// TIA Portal V20 export
DATA_BLOCK "IdentMvHmi"   // DB214
// stored: MemoryReserve 100
   VAR
      unitIdentMv : Array[0.."NO_OF_UNITS"] of "typeEMIdentMv";
   END_VAR
BEGIN
   unitIdentMv[0].identMvEM[0..7].selectedUnit := 0;
   unitIdentMv[0].identMvEM[0..7].selectedEM := 0;
   unitIdentMv[0].identMvEM[0..7].mvReaderId := 0;
   unitIdentMv[0].identMvEM[0..7].numberOfMv := 0;
   unitIdentMv[0].identMvEM[0].mvReader[0..1].deviceName := WSTRING#'';
   unitIdentMv[0].identMvEM[1].mvReader[0..1].deviceName := WSTRING#'';
   unitIdentMv[0].identMvEM[2].mvReader[0..1].deviceName := WSTRING#'';
   unitIdentMv[0].identMvEM[3].mvReader[0..1].deviceName := WSTRING#'';
   unitIdentMv[0].identMvEM[4].mvReader[0..1].deviceName := WSTRING#'';
   unitIdentMv[0].identMvEM[5].mvReader[0..1].deviceName := WSTRING#'';
   unitIdentMv[0].identMvEM[6].mvReader[0..1].deviceName := WSTRING#'';
   unitIdentMv[0].identMvEM[7].mvReader[0..1].deviceName := WSTRING#'';
   unitIdentMv[0].identMvEM[0].mvReader[0..1].deviceType := WSTRING#'';
   unitIdentMv[0].identMvEM[1].mvReader[0..1].deviceType := WSTRING#'';
   unitIdentMv[0].identMvEM[2].mvReader[0..1].deviceType := WSTRING#'';
   unitIdentMv[0].identMvEM[3].mvReader[0..1].deviceType := WSTRING#'';
   unitIdentMv[0].identMvEM[4].mvReader[0..1].deviceType := WSTRING#'';
   unitIdentMv[0].identMvEM[5].mvReader[0..1].deviceType := WSTRING#'';
   unitIdentMv[0].identMvEM[6].mvReader[0..1].deviceType := WSTRING#'';
   unitIdentMv[0].identMvEM[7].mvReader[0..1].deviceType := WSTRING#'';
   unitIdentMv[0].identMvEM[0].mvReader[0..1].deviceId := 0;
   unitIdentMv[0].identMvEM[1].mvReader[0..1].deviceId := 0;
   unitIdentMv[0].identMvEM[2].mvReader[0..1].deviceId := 0;
   unitIdentMv[0].identMvEM[3].mvReader[0..1].deviceId := 0;
   unitIdentMv[0].identMvEM[4].mvReader[0..1].deviceId := 0;
   unitIdentMv[0].identMvEM[5].mvReader[0..1].deviceId := 0;
   unitIdentMv[0].identMvEM[6].mvReader[0..1].deviceId := 0;
   unitIdentMv[0].identMvEM[7].mvReader[0..1].deviceId := 0;
   unitIdentMv[0].identMvEM[0].mvReader[0..1].tagType := WSTRING#'';
   unitIdentMv[0].identMvEM[1].mvReader[0..1].tagType := WSTRING#'';
   unitIdentMv[0].identMvEM[2].mvReader[0..1].tagType := WSTRING#'';
   unitIdentMv[0].identMvEM[3].mvReader[0..1].tagType := WSTRING#'';
   unitIdentMv[0].identMvEM[4].mvReader[0..1].tagType := WSTRING#'';
   unitIdentMv[0].identMvEM[5].mvReader[0..1].tagType := WSTRING#'';
   unitIdentMv[0].identMvEM[6].mvReader[0..1].tagType := WSTRING#'';
   unitIdentMv[0].identMvEM[7].mvReader[0..1].tagType := WSTRING#'';
   unitIdentMv[0].identMvEM[0].mvReader[0..1].cameraMode := WSTRING#'';
   unitIdentMv[0].identMvEM[1].mvReader[0..1].cameraMode := WSTRING#'';
   unitIdentMv[0].identMvEM[2].mvReader[0..1].cameraMode := WSTRING#'';
   unitIdentMv[0].identMvEM[3].mvReader[0..1].cameraMode := WSTRING#'';
   unitIdentMv[0].identMvEM[4].mvReader[0..1].cameraMode := WSTRING#'';
   unitIdentMv[0].identMvEM[5].mvReader[0..1].cameraMode := WSTRING#'';
   unitIdentMv[0].identMvEM[6].mvReader[0..1].cameraMode := WSTRING#'';
   unitIdentMv[0].identMvEM[7].mvReader[0..1].cameraMode := WSTRING#'';
   unitIdentMv[0].identMvEM[0].mvReader[0..1].resultState := WSTRING#'';
   unitIdentMv[0].identMvEM[1].mvReader[0..1].resultState := WSTRING#'';
   unitIdentMv[0].identMvEM[2].mvReader[0..1].resultState := WSTRING#'';
   unitIdentMv[0].identMvEM[3].mvReader[0..1].resultState := WSTRING#'';
   unitIdentMv[0].identMvEM[4].mvReader[0..1].resultState := WSTRING#'';
   unitIdentMv[0].identMvEM[5].mvReader[0..1].resultState := WSTRING#'';
   unitIdentMv[0].identMvEM[6].mvReader[0..1].resultState := WSTRING#'';
   unitIdentMv[0].identMvEM[7].mvReader[0..1].resultState := WSTRING#'';
   unitIdentMv[0].identMvEM[0].mvReader[0..1].progNo := 0;
   unitIdentMv[0].identMvEM[1].mvReader[0..1].progNo := 0;
   unitIdentMv[0].identMvEM[2].mvReader[0..1].progNo := 0;
   unitIdentMv[0].identMvEM[3].mvReader[0..1].progNo := 0;
   unitIdentMv[0].identMvEM[4].mvReader[0..1].progNo := 0;
   unitIdentMv[0].identMvEM[5].mvReader[0..1].progNo := 0;
   unitIdentMv[0].identMvEM[6].mvReader[0..1].progNo := 0;
   unitIdentMv[0].identMvEM[7].mvReader[0..1].progNo := 0;
   unitIdentMv[0].identMvEM[0].mvReader[0..1].progNumberWrite := 0;
   unitIdentMv[0].identMvEM[1].mvReader[0..1].progNumberWrite := 0;
   unitIdentMv[0].identMvEM[2].mvReader[0..1].progNumberWrite := 0;
   unitIdentMv[0].identMvEM[3].mvReader[0..1].progNumberWrite := 0;
   unitIdentMv[0].identMvEM[4].mvReader[0..1].progNumberWrite := 0;
   unitIdentMv[0].identMvEM[5].mvReader[0..1].progNumberWrite := 0;
   unitIdentMv[0].identMvEM[6].mvReader[0..1].progNumberWrite := 0;
   unitIdentMv[0].identMvEM[7].mvReader[0..1].progNumberWrite := 0;
   unitIdentMv[0].identMvEM[0].mvReader[0..1].pushbutton := 16#0000;
   unitIdentMv[0].identMvEM[1].mvReader[0..1].pushbutton := 16#0000;
   unitIdentMv[0].identMvEM[2].mvReader[0..1].pushbutton := 16#0000;
   unitIdentMv[0].identMvEM[3].mvReader[0..1].pushbutton := 16#0000;
   unitIdentMv[0].identMvEM[4].mvReader[0..1].pushbutton := 16#0000;
   unitIdentMv[0].identMvEM[5].mvReader[0..1].pushbutton := 16#0000;
   unitIdentMv[0].identMvEM[6].mvReader[0..1].pushbutton := 16#0000;
   unitIdentMv[0].identMvEM[7].mvReader[0..1].pushbutton := 16#0000;
   unitIdentMv[0].identMvEM[0].mvReader[0..1].enablePushbutton := 16#0000;
   unitIdentMv[0].identMvEM[1].mvReader[0..1].enablePushbutton := 16#0000;
   unitIdentMv[0].identMvEM[2].mvReader[0..1].enablePushbutton := 16#0000;
   unitIdentMv[0].identMvEM[3].mvReader[0..1].enablePushbutton := 16#0000;
   unitIdentMv[0].identMvEM[4].mvReader[0..1].enablePushbutton := 16#0000;
   unitIdentMv[0].identMvEM[5].mvReader[0..1].enablePushbutton := 16#0000;
   unitIdentMv[0].identMvEM[6].mvReader[0..1].enablePushbutton := 16#0000;
   unitIdentMv[0].identMvEM[7].mvReader[0..1].enablePushbutton := 16#0000;
   unitIdentMv[0].identMvEM[0].mvReader[0..1].status := 16#0000;
   unitIdentMv[0].identMvEM[1].mvReader[0..1].status := 16#0000;
   unitIdentMv[0].identMvEM[2].mvReader[0..1].status := 16#0000;
   unitIdentMv[0].identMvEM[3].mvReader[0..1].status := 16#0000;
   unitIdentMv[0].identMvEM[4].mvReader[0..1].status := 16#0000;
   unitIdentMv[0].identMvEM[5].mvReader[0..1].status := 16#0000;
   unitIdentMv[0].identMvEM[6].mvReader[0..1].status := 16#0000;
   unitIdentMv[0].identMvEM[7].mvReader[0..1].status := 16#0000;
   unitIdentMv[0].identMvEM[0].mvReader[0..1].alarmCategorie := 0;
   unitIdentMv[0].identMvEM[1].mvReader[0..1].alarmCategorie := 0;
   unitIdentMv[0].identMvEM[2].mvReader[0..1].alarmCategorie := 0;
   unitIdentMv[0].identMvEM[3].mvReader[0..1].alarmCategorie := 0;
   unitIdentMv[0].identMvEM[4].mvReader[0..1].alarmCategorie := 0;
   unitIdentMv[0].identMvEM[5].mvReader[0..1].alarmCategorie := 0;
   unitIdentMv[0].identMvEM[6].mvReader[0..1].alarmCategorie := 0;
   unitIdentMv[0].identMvEM[7].mvReader[0..1].alarmCategorie := 0;
   unitIdentMv[0].identMvEM[0].mvReader[0..1].alarmNo := 0;
   unitIdentMv[0].identMvEM[1].mvReader[0..1].alarmNo := 0;
   unitIdentMv[0].identMvEM[2].mvReader[0..1].alarmNo := 0;
   unitIdentMv[0].identMvEM[3].mvReader[0..1].alarmNo := 0;
   unitIdentMv[0].identMvEM[4].mvReader[0..1].alarmNo := 0;
   unitIdentMv[0].identMvEM[5].mvReader[0..1].alarmNo := 0;
   unitIdentMv[0].identMvEM[6].mvReader[0..1].alarmNo := 0;
   unitIdentMv[0].identMvEM[7].mvReader[0..1].alarmNo := 0;
   unitIdentMv[0].identMvEM[0].mvReader[0..1].alarmCode := 16#0000_0000;
   unitIdentMv[0].identMvEM[1].mvReader[0..1].alarmCode := 16#0000_0000;
   unitIdentMv[0].identMvEM[2].mvReader[0..1].alarmCode := 16#0000_0000;
   unitIdentMv[0].identMvEM[3].mvReader[0..1].alarmCode := 16#0000_0000;
   unitIdentMv[0].identMvEM[4].mvReader[0..1].alarmCode := 16#0000_0000;
   unitIdentMv[0].identMvEM[5].mvReader[0..1].alarmCode := 16#0000_0000;
   unitIdentMv[0].identMvEM[6].mvReader[0..1].alarmCode := 16#0000_0000;
   unitIdentMv[0].identMvEM[7].mvReader[0..1].alarmCode := 16#0000_0000;
   unitIdentMv[0].identMvEM[0].mvReader[0..1].resultColor := 0;
   unitIdentMv[0].identMvEM[1].mvReader[0..1].resultColor := 0;
   unitIdentMv[0].identMvEM[2].mvReader[0..1].resultColor := 0;
   unitIdentMv[0].identMvEM[3].mvReader[0..1].resultColor := 0;
   unitIdentMv[0].identMvEM[4].mvReader[0..1].resultColor := 0;
   unitIdentMv[0].identMvEM[5].mvReader[0..1].resultColor := 0;
   unitIdentMv[0].identMvEM[6].mvReader[0..1].resultColor := 0;
   unitIdentMv[0].identMvEM[7].mvReader[0..1].resultColor := 0;
   unitIdentMv[0].identMvEM[0].mvReader[0..1].statusColorCode := 0;
   unitIdentMv[0].identMvEM[1].mvReader[0..1].statusColorCode := 0;
   unitIdentMv[0].identMvEM[2].mvReader[0..1].statusColorCode := 0;
   unitIdentMv[0].identMvEM[3].mvReader[0..1].statusColorCode := 0;
   unitIdentMv[0].identMvEM[4].mvReader[0..1].statusColorCode := 0;
   unitIdentMv[0].identMvEM[5].mvReader[0..1].statusColorCode := 0;
   unitIdentMv[0].identMvEM[6].mvReader[0..1].statusColorCode := 0;
   unitIdentMv[0].identMvEM[7].mvReader[0..1].statusColorCode := 0;
   unitIdentMv[0].identMvEM[0].mvReader[0..1].datRead1 := '';
   unitIdentMv[0].identMvEM[1].mvReader[0..1].datRead1 := '';
   unitIdentMv[0].identMvEM[2].mvReader[0..1].datRead1 := '';
   unitIdentMv[0].identMvEM[3].mvReader[0..1].datRead1 := '';
   unitIdentMv[0].identMvEM[4].mvReader[0..1].datRead1 := '';
   unitIdentMv[0].identMvEM[5].mvReader[0..1].datRead1 := '';
   unitIdentMv[0].identMvEM[6].mvReader[0..1].datRead1 := '';
   unitIdentMv[0].identMvEM[7].mvReader[0..1].datRead1 := '';
   unitIdentMv[0].identMvEM[0].mvReader[0..1].datRead2 := '';
   unitIdentMv[0].identMvEM[1].mvReader[0..1].datRead2 := '';
   unitIdentMv[0].identMvEM[2].mvReader[0..1].datRead2 := '';
   unitIdentMv[0].identMvEM[3].mvReader[0..1].datRead2 := '';
   unitIdentMv[0].identMvEM[4].mvReader[0..1].datRead2 := '';
   unitIdentMv[0].identMvEM[5].mvReader[0..1].datRead2 := '';
   unitIdentMv[0].identMvEM[6].mvReader[0..1].datRead2 := '';
   unitIdentMv[0].identMvEM[7].mvReader[0..1].datRead2 := '';
   unitIdentMv[0].identMvEM[0].mvReader[0..1].datRead3 := '';
   unitIdentMv[0].identMvEM[1].mvReader[0..1].datRead3 := '';
   unitIdentMv[0].identMvEM[2].mvReader[0..1].datRead3 := '';
   unitIdentMv[0].identMvEM[3].mvReader[0..1].datRead3 := '';
   unitIdentMv[0].identMvEM[4].mvReader[0..1].datRead3 := '';
   unitIdentMv[0].identMvEM[5].mvReader[0..1].datRead3 := '';
   unitIdentMv[0].identMvEM[6].mvReader[0..1].datRead3 := '';
   unitIdentMv[0].identMvEM[7].mvReader[0..1].datRead3 := '';
   unitIdentMv[0].identMvEM[0].mvReader[0..1].datRead4 := '';
   unitIdentMv[0].identMvEM[1].mvReader[0..1].datRead4 := '';
   unitIdentMv[0].identMvEM[2].mvReader[0..1].datRead4 := '';
   unitIdentMv[0].identMvEM[3].mvReader[0..1].datRead4 := '';
   unitIdentMv[0].identMvEM[4].mvReader[0..1].datRead4 := '';
   unitIdentMv[0].identMvEM[5].mvReader[0..1].datRead4 := '';
   unitIdentMv[0].identMvEM[6].mvReader[0..1].datRead4 := '';
   unitIdentMv[0].identMvEM[7].mvReader[0..1].datRead4 := '';
   unitIdentMv[0].identMvEM[0].mvReader[0].datWrite1 := '';
   unitIdentMv[0].identMvEM[0].mvReader[1].datWrite1 := 'Siemens';
   unitIdentMv[0].identMvEM[1].mvReader[0..1].datWrite1 := '';
   unitIdentMv[0].identMvEM[2].mvReader[0..1].datWrite1 := '';
   unitIdentMv[0].identMvEM[3].mvReader[0..1].datWrite1 := '';
   unitIdentMv[0].identMvEM[4].mvReader[0..1].datWrite1 := '';
   unitIdentMv[0].identMvEM[5].mvReader[0..1].datWrite1 := '';
   unitIdentMv[0].identMvEM[6].mvReader[0..1].datWrite1 := '';
   unitIdentMv[0].identMvEM[7].mvReader[0..1].datWrite1 := '';
   unitIdentMv[0].identMvEM[0].mvReader[0..1].datWrite2 := '';
   unitIdentMv[0].identMvEM[1].mvReader[0..1].datWrite2 := '';
   unitIdentMv[0].identMvEM[2].mvReader[0..1].datWrite2 := '';
   unitIdentMv[0].identMvEM[3].mvReader[0..1].datWrite2 := '';
   unitIdentMv[0].identMvEM[4].mvReader[0..1].datWrite2 := '';
   unitIdentMv[0].identMvEM[5].mvReader[0..1].datWrite2 := '';
   unitIdentMv[0].identMvEM[6].mvReader[0..1].datWrite2 := '';
   unitIdentMv[0].identMvEM[7].mvReader[0..1].datWrite2 := '';
   unitIdentMv[0].identMvEM[0].mvReader[0..1].datWrite3 := '';
   unitIdentMv[0].identMvEM[1].mvReader[0..1].datWrite3 := '';
   unitIdentMv[0].identMvEM[2].mvReader[0..1].datWrite3 := '';
   unitIdentMv[0].identMvEM[3].mvReader[0..1].datWrite3 := '';
   unitIdentMv[0].identMvEM[4].mvReader[0..1].datWrite3 := '';
   unitIdentMv[0].identMvEM[5].mvReader[0..1].datWrite3 := '';
   unitIdentMv[0].identMvEM[6].mvReader[0..1].datWrite3 := '';
   unitIdentMv[0].identMvEM[7].mvReader[0..1].datWrite3 := '';
   unitIdentMv[0].identMvEM[0].mvReader[0..1].datWrite4 := '';
   unitIdentMv[0].identMvEM[1].mvReader[0..1].datWrite4 := '';
   unitIdentMv[0].identMvEM[2].mvReader[0..1].datWrite4 := '';
   unitIdentMv[0].identMvEM[3].mvReader[0..1].datWrite4 := '';
   unitIdentMv[0].identMvEM[4].mvReader[0..1].datWrite4 := '';
   unitIdentMv[0].identMvEM[5].mvReader[0..1].datWrite4 := '';
   unitIdentMv[0].identMvEM[6].mvReader[0..1].datWrite4 := '';
   unitIdentMv[0].identMvEM[7].mvReader[0..1].datWrite4 := '';
END_DATA_BLOCK
